INTERFACE I_LoggerConfigBuilder

// Applies the configuration
METHOD Apply
VAR_INPUT
	writeConfigToLog	: BOOL;	// Will write applied configuration to the target log file if set to TRUE
END_VAR
END_METHOD

(* Set the time after which the logs will be deleted.*)
METHOD DeleteLogsAfter : I_LoggerConfigBuilder
VAR_INPUT
	days			: UINT;	// Delete log files after X - days
	checkInterval	: TIME;	// Check interval for deleting the existing files
END_VAR
END_METHOD

(* Sets the log file extension <file>.<extension>. 
You can or can't include the dot, it will be checked and added either way.*)
METHOD SetLogExtension : I_LoggerConfigBuilder
VAR_INPUT
	extension	: STRING;
END_VAR
END_METHOD

// Sets the log file name
METHOD SetLogFileName : I_LoggerConfigBuilder
VAR_INPUT
	name	: STRING;
END_VAR
END_METHOD

// Sets the path where the logs will be stored.
METHOD SetLogFilePath : I_LoggerConfigBuilder
VAR_INPUT
	path	: Tc2_System.T_MaxString;
END_VAR
END_METHOD

// Sets the NetId of the device where logs will be stored.
METHOD SetNetId : I_LoggerConfigBuilder
VAR_INPUT
	netId	: Tc2_System.T_AmsNetID;
END_VAR
END_METHOD

// Sets the rolling interval (in hours) - how offten new log file is created. If set to 0, a single file is created. Beware of DeleteCheckInterval, which will delete this file and you will lose these files in that case.
METHOD SetRollingInterval : I_LoggerConfigBuilder
VAR_INPUT
	hours	: UINT;
END_VAR
END_METHOD

END_INTERFACE

(* stored: Version 1.1.0.1, ProductVersion 3.1.4024.14
   Itf I_LoggerConfigBuilder: Id {bb42e3f5-3123-09b0-0e7d-84e61a15a959}
   Method Apply: Id {97b282f8-4249-0806-190f-9a4e82bfb32f}
   Method DeleteLogsAfter: Id {87176372-6c90-0804-3b4f-9d37315855a8}
   Method SetLogExtension: Id {a5817c73-770b-028d-3b79-475c96629825}
   Method SetLogFileName: Id {bfeddf5b-961c-02b2-325a-3bfda6762abd}
   Method SetLogFilePath: Id {f3a0e5f9-adae-06f0-237b-ca900dbcd9e8}
   Method SetNetId: Id {25ffe7e2-0c70-015d-20a2-435e9afb4a50}
   Method SetRollingInterval: Id {f57fa4b1-bfad-046f-178c-8ce37acdf01a} *)
